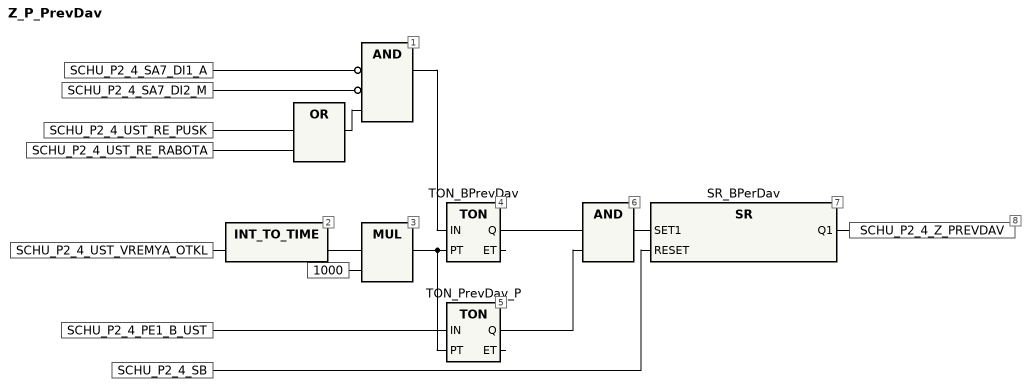
[picture p288: Z_P_PrevDav (CFC)]
_CFC_ (* Continuous Function Chart, elements in execution order *)
#0 OR(SCHU_P2_4_UST_RE_PUSK, SCHU_P2_4_UST_RE_RABOTA)
#1 AND(NOT SCHU_P2_4_SA7_DI1_A, NOT SCHU_P2_4_SA7_DI2_M, #0)
#2 INT_TO_TIME(SCHU_P2_4_UST_VREMYA_OTKL)
#3 MUL(#2, 1000)
#4 TON_BPrevDav:TON(IN: #1, PT: #3)
#5 TON_PrevDav_P:TON(IN: SCHU_P2_4_PE1_B_UST, PT: #3)
#6 AND(#4.Q, #5.Q)
#7 SR_BPerDav:SR(SET1: #6, RESET: SCHU_P2_4_SB)
#8 SCHU_P2_4_Z_PREVDAV <= #7.Q1
_END_CFC_
(* the same logic as Structured Text *)
_t30 := INT_TO_TIME(SCHU_P2_4_UST_VREMYA_OTKL) * 1000;
TON_BPrevDav(IN := NOT SCHU_P2_4_SA7_DI1_A AND NOT SCHU_P2_4_SA7_DI2_M AND (SCHU_P2_4_UST_RE_PUSK OR SCHU_P2_4_UST_RE_RABOTA), PT := _t30);
TON_PrevDav_P(IN := SCHU_P2_4_PE1_B_UST, PT := _t30);
SR_BPerDav(SET1 := TON_BPrevDav.Q AND TON_PrevDav_P.Q, RESET := SCHU_P2_4_SB);
SCHU_P2_4_Z_PREVDAV := SR_BPerDav.Q1;
END_PROGRAM

(* POU TZBiS/TZB/Sbros_All, CFC *)
PROGRAM Sbros_All
VAR
END_VAR
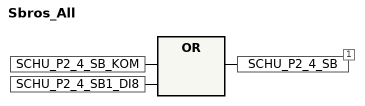
_CFC_ (* Continuous Function Chart, elements in execution order *)
#0 OR(SCHU_P2_4_SB_KOM, SCHU_P2_4_SB1_DI8)
#1 SCHU_P2_4_SB <= #0
_END_CFC_
(* the same logic as Structured Text *)
SCHU_P2_4_SB := SCHU_P2_4_SB_KOM OR SCHU_P2_4_SB1_DI8;
END_PROGRAM

(* POU TZBiS/TZB/Z_Pozhar, CFC *)
PROGRAM Z_Pozhar
VAR
	SR_Pozhar: SR;
END_VAR
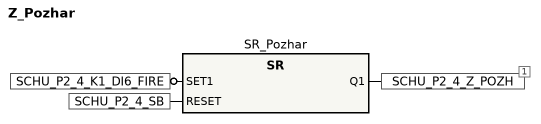
_CFC_ (* Continuous Function Chart, elements in execution order *)
#0 SR_Pozhar:SR(SET1: NOT SCHU_P2_4_K1_DI6_FIRE, RESET: SCHU_P2_4_SB)
#1 SCHU_P2_4_Z_POZH <= #0.Q1
_END_CFC_
(* the same logic as Structured Text *)
SR_Pozhar(SET1 := NOT SCHU_P2_4_K1_DI6_FIRE, RESET := SCHU_P2_4_SB);
SCHU_P2_4_Z_POZH := SR_Pozhar.Q1;
END_PROGRAM

(* POU TZBiS/TZB/Z_YA1_Otk, CFC *)
PROGRAM Z_YA1_Otk
VAR
	SR_YA1_Otkaz: SR;
	TON_YA1_Otk: TON;
	TON_YA1_N_OTKR: TON;
	TON_YA1_N_ZAKR: TON;
	TON_YA1_ZKR: TON;
	TON_AVT: TON;

	a: BOOL;
	b: BOOL;
	c: BOOL;
	d: BOOL;
	e: BOOL;
END_VAR
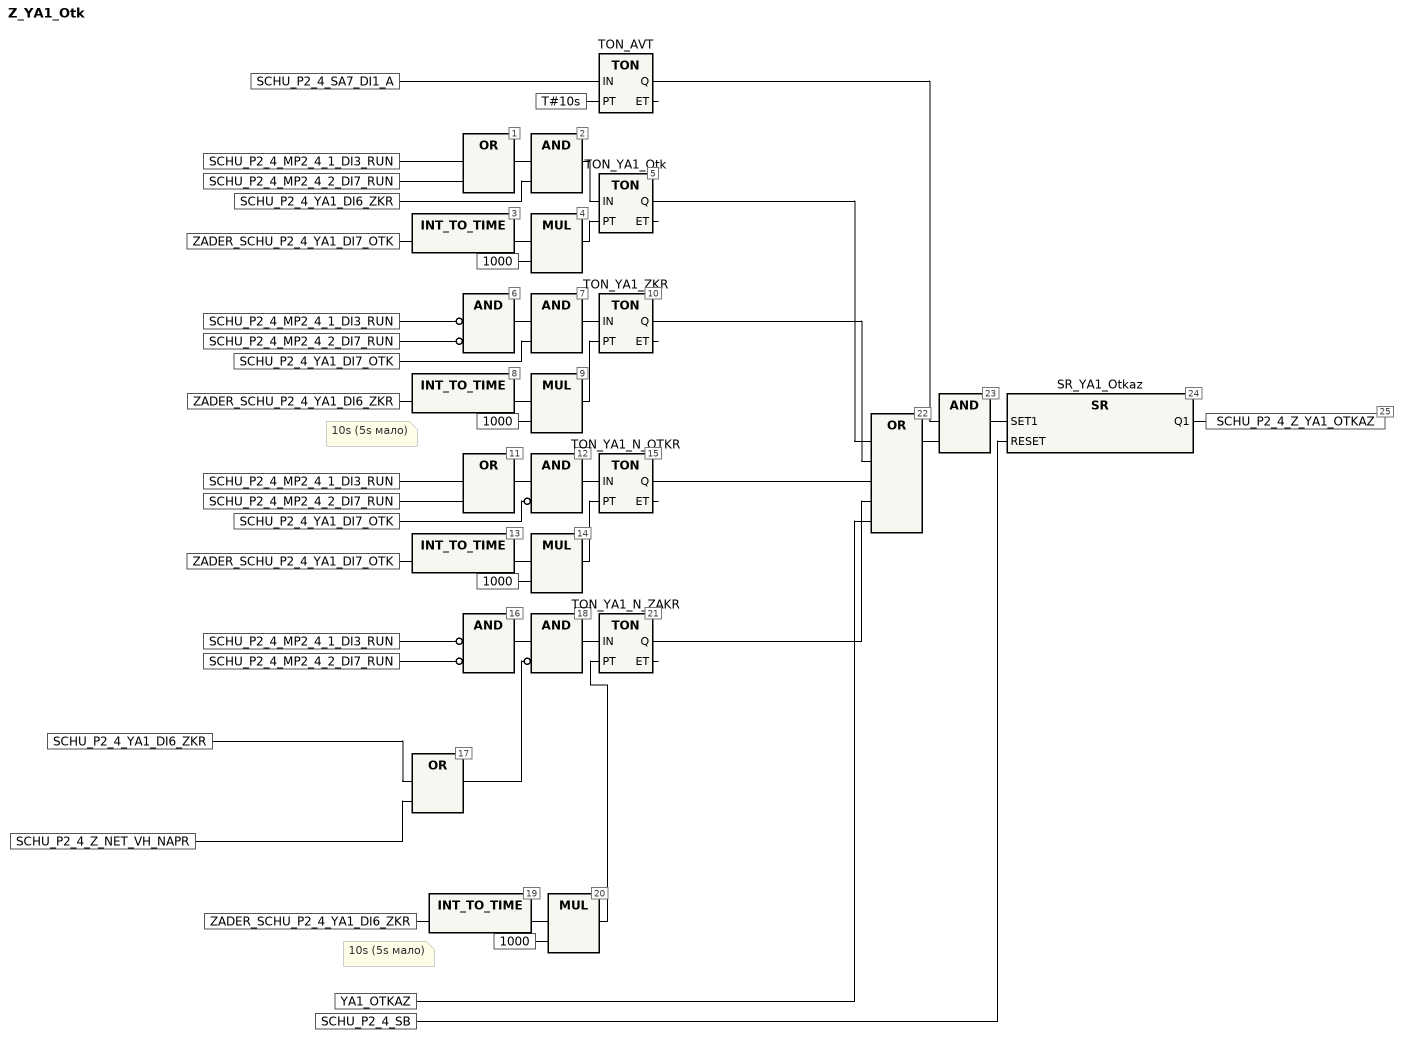
_CFC_ (* Continuous Function Chart, elements in execution order *)
(* 10s (5s мало) *)
(* 10s (5s мало) *)
#0 TON_AVT:TON(IN: SCHU_P2_4_SA7_DI1_A, PT: T#10s)
#1 OR(SCHU_P2_4_MP2_4_1_DI3_RUN, SCHU_P2_4_MP2_4_2_DI7_RUN)
#2 AND(#1, SCHU_P2_4_YA1_DI6_ZKR)
#3 INT_TO_TIME(ZADER_SCHU_P2_4_YA1_DI7_OTK)
#4 MUL(#3, 1000)
#5 TON_YA1_Otk:TON(IN: #2, PT: #4)
#6 AND(NOT SCHU_P2_4_MP2_4_1_DI3_RUN, NOT SCHU_P2_4_MP2_4_2_DI7_RUN)
#7 AND(#6, SCHU_P2_4_YA1_DI7_OTK)
#8 INT_TO_TIME(ZADER_SCHU_P2_4_YA1_DI6_ZKR)
#9 MUL(#8, 1000)
#10 TON_YA1_ZKR:TON(IN: #7, PT: #9)
#11 OR(SCHU_P2_4_MP2_4_1_DI3_RUN, SCHU_P2_4_MP2_4_2_DI7_RUN)
#12 AND(#11, NOT SCHU_P2_4_YA1_DI7_OTK)
#13 INT_TO_TIME(ZADER_SCHU_P2_4_YA1_DI7_OTK)
#14 MUL(#13, 1000)
#15 TON_YA1_N_OTKR:TON(IN: #12, PT: #14)
#16 AND(NOT SCHU_P2_4_MP2_4_1_DI3_RUN, NOT SCHU_P2_4_MP2_4_2_DI7_RUN)
#17 OR(SCHU_P2_4_YA1_DI6_ZKR, SCHU_P2_4_Z_NET_VH_NAPR)
#18 AND(#16, NOT #17)
#19 INT_TO_TIME(ZADER_SCHU_P2_4_YA1_DI6_ZKR)
#20 MUL(#19, 1000)
#21 TON_YA1_N_ZAKR:TON(IN: #18, PT: #20)
#22 OR(#5.Q, #10.Q, #15.Q, #21.Q, YA1_OTKAZ)
#23 AND(#0.Q, #22)
#24 SR_YA1_Otkaz:SR(SET1: #23, RESET: SCHU_P2_4_SB)
#25 SCHU_P2_4_Z_YA1_OTKAZ <= #24.Q1
_END_CFC_
(* the same logic as Structured Text *)
(* 10s (5s мало) *)
(* 10s (5s мало) *)
TON_AVT(IN := SCHU_P2_4_SA7_DI1_A, PT := T#10s);
TON_YA1_Otk(IN := (SCHU_P2_4_MP2_4_1_DI3_RUN OR SCHU_P2_4_MP2_4_2_DI7_RUN) AND SCHU_P2_4_YA1_DI6_ZKR, PT := INT_TO_TIME(ZADER_SCHU_P2_4_YA1_DI7_OTK) * 1000);
TON_YA1_ZKR(IN := (NOT SCHU_P2_4_MP2_4_1_DI3_RUN AND NOT SCHU_P2_4_MP2_4_2_DI7_RUN) AND SCHU_P2_4_YA1_DI7_OTK, PT := INT_TO_TIME(ZADER_SCHU_P2_4_YA1_DI6_ZKR) * 1000);
TON_YA1_N_OTKR(IN := (SCHU_P2_4_MP2_4_1_DI3_RUN OR SCHU_P2_4_MP2_4_2_DI7_RUN) AND NOT SCHU_P2_4_YA1_DI7_OTK, PT := INT_TO_TIME(ZADER_SCHU_P2_4_YA1_DI7_OTK) * 1000);
TON_YA1_N_ZAKR(IN := (NOT SCHU_P2_4_MP2_4_1_DI3_RUN AND NOT SCHU_P2_4_MP2_4_2_DI7_RUN) AND NOT (SCHU_P2_4_YA1_DI6_ZKR OR SCHU_P2_4_Z_NET_VH_NAPR), PT := INT_TO_TIME(ZADER_SCHU_P2_4_YA1_DI6_ZKR) * 1000);
SR_YA1_Otkaz(SET1 := TON_AVT.Q AND (TON_YA1_Otk.Q OR TON_YA1_ZKR.Q OR TON_YA1_N_OTKR.Q OR TON_YA1_N_ZAKR.Q OR YA1_OTKAZ), RESET := SCHU_P2_4_SB);
SCHU_P2_4_Z_YA1_OTKAZ := SR_YA1_Otkaz.Q1;
END_PROGRAM

(* POU TZBiS/TZB/Z_YA2_Otk, CFC *)
PROGRAM Z_YA2_Otk
VAR
	SR_YA2_Otk: SR;
	TON_YA2_Rassog: TON;
	RT_Rassog: R_TRIG;
	TON_YA2_Rassog1: TON;
	TIME_DELAY: TIME;
END_VAR
VAR (* helpers for the ST form of the networks *)
	_t14 : BOOL;
END_VAR
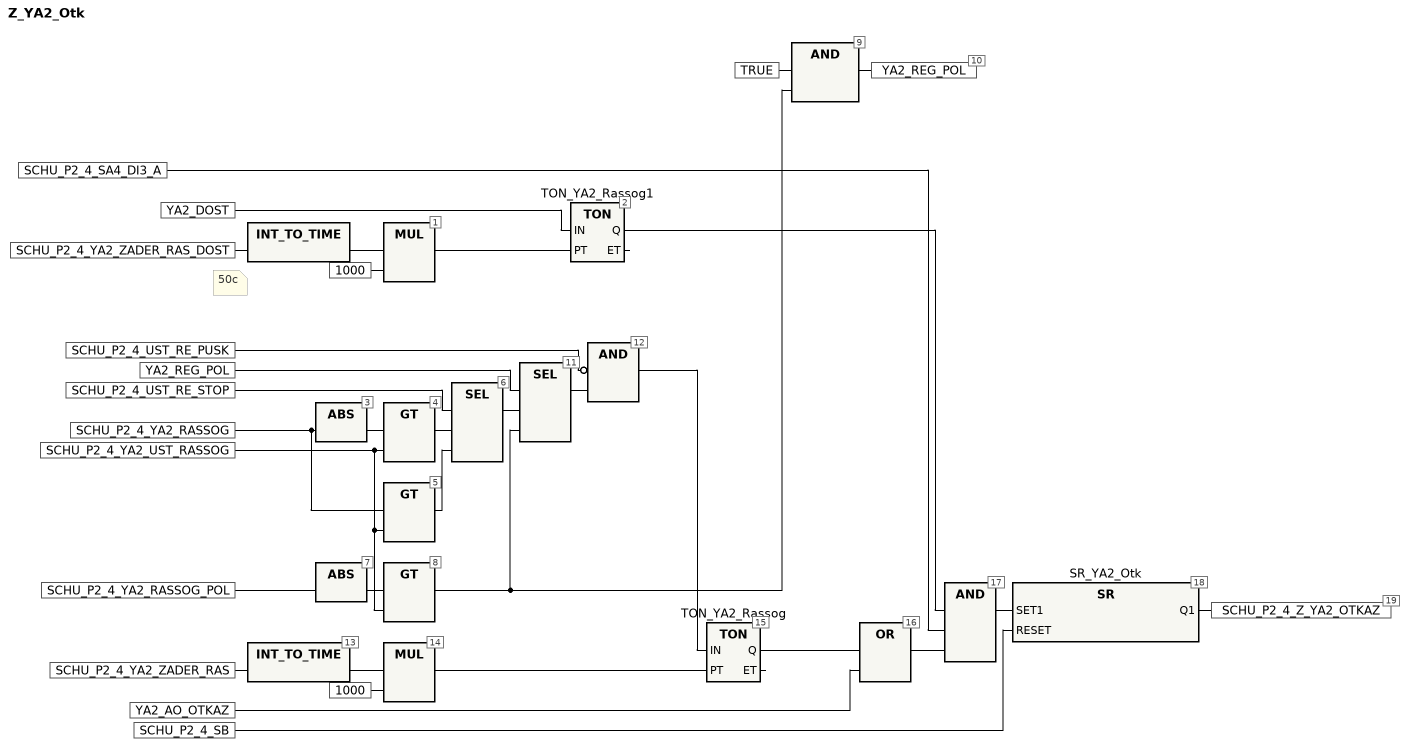
